FUNCTION_BLOCK Tank1
VAR_INPUT
	//bSwitchFill : BOOL;
	bSwitchSink : BOOL;
END_VAR
VAR_IN_OUT
	bSwitchFill : BOOL;
END_VAR
VAR_OUTPUT
END_VAR
VAR
	bShl : BOOL := FALSE;
	bSll : BOOL := TRUE;
	nState : INT;
	level: INT := 5;
	tTime1 : TON;
	tTime2 : TON;
	rTrig1 : R_TRIG;
	rTrig2 : R_TRIG;
	
	
END_VAR


CASE nState OF
	0:	
		
		IF  NOT bSwitchSink THEN
			IF bSll THEN
				bSwitchFill := TRUE;
			END_IF
			tTime1(IN := bSwitchFill,PT := T#2S);
			rTrig1(CLK := tTime1.Q);
			IF rTrig1.Q THEN
				level := level + 1;
				tTime1(IN := FALSE);
				IF level = 100 THEN
				bShl := TRUE;
				bSll := FALSE;	
				bSwitchFill := FALSE;
				nState := 10;
				END_IF
			END_IF
		
 		
		ELSIF  bSwitchSink THEN
			IF bSll THEN
				bSwitchFill := TRUE;
			END_IF
			tTime1(IN := bSwitchFill,PT := T#3S);
			rTrig1(CLK := tTime1.Q);
			IF rTrig1.Q THEN
				level := level + 1;
				tTime1(IN := FALSE);
				IF level = 100 THEN
				bShl := TRUE;
				bSll := FALSE;
				bSwitchFill := FALSE;
				nState := 10;
				END_IF
			END_IF
		END_IF
		
	10: 
		
		IF  bSwitchSink  THEN
			IF bShl AND level > 90 THEN
				bSwitchFill := FALSE;
				tTime2(IN := bSwitchSink,PT := T#1S);
				rTrig2(CLK := tTime2.Q);
				IF rTrig2.q THEN
				tTime2(IN := FALSE);
				level := level - 1;
				IF level = 5 THEN
				bSwitchSink := FALSE;
				bShl := FALSE;
				bSll := TRUE;
				nState := 0;
				END_IF
				END_IF
			ELSIF level <= 90 THEN
					IF bSwitchFill THEN
					
						tTime2(IN := bSwitchSink,PT := T#3S);
						rTrig2(CLK := tTime2.Q);
						IF rTrig2.q THEN
						tTime2(IN := FALSE);
						level := level + 1;
						IF level = 100 THEN
						bSwitchSink := FALSE;
						bShl := TRUE;
						bSll := FALSE;
						nState := 10;
						END_IF
						END_IF
						
					ELSE
						tTime2(IN := bSwitchSink,PT := T#1S);
						rTrig2(CLK := tTime2.Q);
						IF rTrig2.q THEN
						tTime2(IN := FALSE);
						level := level - 1;
						IF level = 5 THEN
						bSwitchSink := FALSE;
						bShl := FALSE;
						bSll := TRUE;
						nState := 0;
						END_IF
						END_IF
						
					END_IF
			
			END_IF		
			
			
		END_IF
		
		
END_CASE

END_FUNCTION_BLOCK

(* stored: Version 1.1.0.1, ProductVersion 3.1.4024.0
   POU Tank1: Id {f642bd64-7535-452f-aba8-a08221a41d03}, SpecialFunc None *)
